FUNCTION_BLOCK MLMODEL (* HEAD COMPUTING cv\ml model *)
  (* Version 1.0, AN, SWDC RTSoft *)
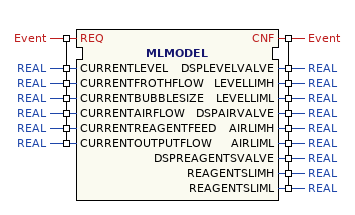
  EVENT_INPUT
    REQ WITH CURRENTLEVEL, CURRENTFROTHFLOW, CURRENTBUBBLESIZE, CURRENTAIRFLOW, CURRENTREAGENTFEED, CURRENTOUTPUTFLOW;
  END_EVENT
  EVENT_OUTPUT
    CNF WITH DSPLEVELVALVE, LEVELLIMH, LEVELLIML, DSPAIRVALVE, AIRLIMH, AIRLIML, DSPREAGENTSVALVE, REAGENTSLIMH, REAGENTSLIML;
  END_EVENT
  VAR_INPUT
    CURRENTLEVEL : REAL;
    CURRENTFROTHFLOW : REAL;
    CURRENTBUBBLESIZE : REAL;
    CURRENTAIRFLOW : REAL;
    CURRENTREAGENTFEED : REAL;
    CURRENTOUTPUTFLOW : REAL;
  END_VAR
  VAR_OUTPUT
    DSPLEVELVALVE : REAL;
    LEVELLIMH : REAL;
    LEVELLIML : REAL;
    DSPAIRVALVE : REAL;
    AIRLIMH : REAL;
    AIRLIML : REAL;
    DSPREAGENTSVALVE : REAL;
    REAGENTSLIMH : REAL;
    REAGENTSLIML : REAL;
  END_VAR
END_FUNCTION_BLOCK
